(* LS Electric XG5000 project: 241008_연습문제8 *)
(* PLC LSPLC *)

PROGRAM NewProgram (* task: 스캔 프로그램 *)
VAR
    INST : TOF;
    P1 AT %IX0.0.0 : BOOL;
    P10 AT %QX0.1.0 : BOOL;
    플리커 : TON;
    플리커1 : TON;
END_VAR

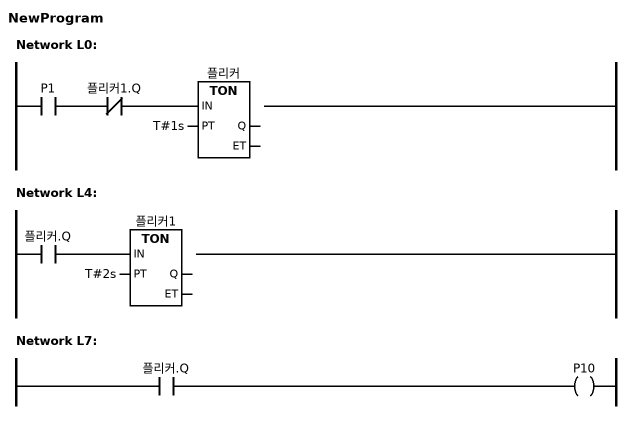
(* Rung L0 *)
플리커(IN := P1 AND NOT 플리커1.Q, PT := T#1s);
(* Rung L4 *)
플리커1(IN := 플리커.Q, PT := T#2s);
(* Rung L7 *)
P10 := 플리커.Q;
END_PROGRAM